// TwinCAT 3 PLC project ButtonControlledGarageDoor
// ProgramVersion: 3.1.4024.0
// libraries:
//   Tc2_Standard, * (Beckhoff Automation GmbH)
//   Tc2_System, * (Beckhoff Automation GmbH)
//   Tc3_Module, * (Beckhoff Automation GmbH)
//   VisuDialogs, * (System)
// project tree:
//   / GlobalTextList.TcGTLO, PlcTask.TcTTO, Visualization Manager.TcVMO (not stored)
//   POUs/ FB_DoorController.TcPOU, FB_BlinkingLight.TcPOU, MAIN.TcPOU
//   VISUs/ Visualization.TcVIS
// real-time tasks:
//   TASK PlcTask: cycle T#10ms, priority 20, ADS port 350

CONFIGURATION ButtonControlledGarageDoor
    RESOURCE PLC ON TwinCAT3
        TASK PlcTask(INTERVAL := T#10ms, PRIORITY := 20);
        PROGRAM MAIN WITH PlcTask : MAIN;
    END_RESOURCE
END_CONFIGURATION

// ---- POUs/MAIN.TcPOU
PROGRAM MAIN
VAR
	fbGarage1 : FB_DoorController;
	bActuation1 : BOOL;
	bOpenButton1 : BOOL;
	bCloseButton1 : BOOL;
	bDriveOverload1 : BOOL; 
	dwLightDelay1 : DWORD := 1000;
	dwBlinkingTimeOn1 : DWORD := 500;
	dwBlinkingTimeOff1 : DWORD := 250;
	bDoorLight1 : BOOL;
	bOpeningLight1 : BOOL;
	bClosingLight1 : BOOL;
	bNoError1 : BOOL;
	sErrorMessage1 : STRING;
	
	fbGarage2 : FB_DoorController;
	bActuation2 : BOOL;
	bOpenButton2 : BOOL;
	bCloseButton2 : BOOL;
	bDriveOverload2 : BOOL; 
	dwLightDelay2 : DWORD := 1000;
	dwBlinkingTimeOn2 : DWORD := 500;
	dwBlinkingTimeOff2 : DWORD := 250;
	bDoorLight2 : BOOL;
	bOpeningLight2 : BOOL;
	bClosingLight2 : BOOL;
	bNoError2 : BOOL;
	sErrorMessage2 : STRING;
END_VAR

fbGarage1(bActuation := bActuation1, 
		  bOpenButton := bOpenButton1, 
		  bCloseButton := bCloseButton1, 
		  bDriveOverload := bDriveOverload1,
		  dwLightDelay := dwLightDelay1,
		  dwBlinkingTimeOn := dwBlinkingTimeOn1,
		  dwBlinkingTimeOff := dwBlinkingTimeOff1,
		  bDoorLight => bDoorLight1, 
		  bOpeningLight => bOpeningLight1, 
		  bClosingLight => bClosingLight1,
		  bNoError => bNoError1,
		  sErrorMessage => sErrorMessage1); 
		  
fbGarage2(bActuation := bActuation2, 
		  bOpenButton := bOpenButton2, 
		  bCloseButton := bCloseButton2, 
		  bDriveOverload := bDriveOverload2,
		  dwLightDelay := dwLightDelay2,
		  dwBlinkingTimeOn := dwBlinkingTimeOn2,
		  dwBlinkingTimeOff := dwBlinkingTimeOff2,
		  bDoorLight => bDoorLight2, 
		  bOpeningLight => bOpeningLight2, 
		  bClosingLight => bClosingLight2,
		  bNoError => bNoError2,
		  sErrorMessage => sErrorMessage2);

END_PROGRAM

// ---- POUs/FB_DoorController.TcPOU
FUNCTION_BLOCK FB_DoorController
VAR_INPUT
	// Button that starts the door
	bActuation : BOOL;
	
	// Buttons that open / close the door respectively
	bOpenButton: BOOL;
	bCloseButton : BOOL;
	
	// Button that makes the door go into a drive overload
	bDriveOverload : BOOL;
	
	// How much time (in ms) should pass in order for the light to turn off when the door has opened / closed 
	dwLightDelay : DWORD;
	
	// On/off times (in miliseconds) for when the garage door light is blinking in state of error
	dwBlinkingTimeOn : DWORD;
	dwBlinkingTimeOff : DWORD;
END_VAR
VAR_OUTPUT
	// Outputs sent to actuators stating that the door is moving up / down
	bDoorUp : BOOL;
	bDoorDown : BOOL;
	
	// Indicates whether the door light should be on or off
	bDoorLight : BOOL;
	
	// Lights that turn on if the door is opened / closed
	bOpeningLight : BOOL;
	bClosingLight : BOOL;
	
	// Variable that'll tell me if I'm in an error state or not
	bNoError : BOOL := TRUE;
	// Displaying a message according to the error we are encountering
	sErrorMessage : STRING;
END_VAR
VAR
	// Variables stating whether the door is opened or closed
	bDoorOpen : BOOL;
	bDoorClosed : BOOL := TRUE;	// Assumption that in the beginning the door is closed
	
	// TRUE when the process was paused during opening / closing
	bPauseWhenOpening : BOOL;
	bPauseWhenClosing : BOOL;

	(* Timer needed for turning the door light off after a certain period of time passes 
	after the door has been opened / closed *)
	fbLightTimer : TON;
	
	// Trigger functions to deal with bouncing
	fbActuation : R_TRIG;
	fbOpenButton : R_TRIG;
	fbCloseButton : R_TRIG;
	fbDriveOverloadButton : R_TRIG;
	
	(* Instance of the BlinkingLight FB needed for the blinking of the actuation button 
	when it goes to an error state *)
	fbBlinkingLight : FB_BlinkingLight;
	
	// Variable needed for initializing the CASE structure states
	nCurrentState : DINT;
	
	// Variables stating which errors we are encountering
	bDriveError : BOOL;
	bOpenError : BOOL; 
	bCloseError : BOOL;
	
	(* Temporary variable that helps me overcome a problem I'm facing due to
	   bOpenButton and bCloseButton being tappers *)
	bPom : BOOL;
	
	// Variables needed only for the visualisation
	Rect1 : BOOL;
	Rect2 : BOOL;

END_VAR

(* This FB is intended to manage the operation of a garage door. It processes inputs
   from various buttons (bActuation, bOpenButton, bCloseButton) and it handles drive
   overloads (bDriveOverload). The block controls the movement of the door (bDoorUp,
   bDoorDown), the activation of lights (bDoorLight, bOpeningLight, bClosingLight),
   and transitions between different states (idle, opening, closing, error). The FB
   also manages the timing for the door's lights, espeially when they need to blink
   in case of errors. Additionally, it tracks whether the door is fully opened or
   fully closed, handles pauses during opening or closing, and displays error messages
   when needed. *)

// Rising edge logic in order to stop bouncing (the signal persisting longer than intended)
fbActuation(CLK := bActuation);
bActuation := fbActuation.Q;
fbOpenButton(CLK := bOpenButton);
bOpenButton := fbOpenButton.Q;
fbCloseButton(CLK := bCloseButton);
bCloseButton := fbCloseButton.Q;
fbDriveOverloadButton(CLK := bDriveOverload);
bDriveOverload := fbDriveOverloadButton.Q;

CASE nCurrentState OF
	
	0:	// Idle
	(* The door is at rest. If the actuation button is pressed, the door either opens 
	   (if closed) or closes (if open). It also checks for a drive overload to 
	   transition into an error state. *)
	
	// If the overload sensor is activated, go to the error state
	IF bDriveOverload THEN
		nCurrentState := 999;
	END_IF
	
	// Reseting
	fbLightTimer.IN := FALSE;
	bDoorLight := FALSE;
	bOpeningLight := FALSE;
	bClosingLight := FALSE;
	
	// If the actuation button is pressed and the door is closed -> open it
	IF bActuation AND (bDoorClosed OR bPauseWhenClosing) THEN
		nCurrentState := 100;
	// If the actuation button is pressed and the door is opened -> close it
	ELSIF bActuation AND (bDoorOpen OR bPauseWhenOpening) THEN
		nCurrentState := 200;
	END_IF
	
	100:	// Opening
	(* The door is moving upwards. It activates the appropriate light and monitors for
	   errors like drive overload or the close button being pressed. If the door reaches 
	   the fully open position, it sets the bDoorOpen flag to TRUE, stops the opening 
	   process, and returns to the idle state. If an error occurs, it pauses the opening 
	   and transitions to the error state. *)
	
	(* If the overload sensor is activated or if the close button is pressed, go to the error state. 
	   bPauseWhenClosing is true because I want to continue with opening after I get out of the error state *)
	IF bDriveOverload OR bCloseButton THEN
		IF bDriveOverload THEN
			bdriveError := TRUE;	
		ELSIF bCloseButton THEN
			bCloseError := TRUE;
		END_IF
		
		bPauseWhenOpening := FALSE;
		bPauseWhenClosing := TRUE;
		nCurrentState := 999;
	END_IF
	
	// RESET EVERYTHING THAT'S GOTTA DO WITH CLOSING HERE
	bDoorDown := FALSE;
	bDoorClosed := FALSE;
	
	// State that the door should go up and turn the light on
	bDoorUp := TRUE;
	bDoorLight := TRUE;
	bOpeningLight := TRUE;
	
	// Code needed only for the visualisation
	Rect1 := TRUE;
	
	// Logic for opening
	IF bOpenButton OR bPom THEN	
		bPom := TRUE;
		bDoorOpen := TRUE;
		bPauseWhenClosing := FALSE;
		bOpeningLight := FALSE;
		
		Rect2 := TRUE;	// Needed only for the visualization
		
		fbLightTimer.IN := TRUE;
		IF fbLightTimer.Q THEN
			bPom := FALSE;
			bDoorLight := FALSE;
			nCurrentState := 0;
		END_IF		
	END_IF
	
	// The opening is paused -> go to idle state
	IF bActuation THEN
		bPauseWhenOpening := TRUE;
		bPauseWhenClosing := FALSE;
		bOpeningLight := FALSE;
	END_IF
	
	IF bPauseWhenOpening THEN
		fbLightTimer.IN := TRUE;
			IF fbLightTimer.Q THEN
				bDoorLight := FALSE;
				nCurrentState := 0;
			END_IF
	END_IF
	
	200:	// Closing
	(* The door is moving downwards. It manages the closing light and checks for errors
	   such as the open button being pressed or a drive overload. If the door reaches the 
	   fully closed position, it sets the bDoorClosed flag to TRUE, stops the closing 
	   process, and returns to the idle state. Similar to the opening state, any error 
	   pauses the closing process and transitions to the error state. *)
	
	(* If the overload sensor is activated or if the open button is pressed, go to the error state. 
	   bPauseWhenOpening is true because I want to continue with closing after I get out of the error state *)
	IF bDriveOverload OR bOpenButton THEN
		IF bDriveOverload THEN
			bdriveError := TRUE;	
		ELSIF bOpenButton THEN
			bOpenError := TRUE;
		END_IF
		
		bPauseWhenOpening := TRUE;
		bPauseWhenClosing := FALSE;
		nCurrentState := 999;
	END_IF
	
	// RESET EVERYTHING THAT'S GOTTA DO WITH OPENING HERE
	bDoorUp := FALSE;
	bDoorOpen := FALSE;
	
	// State that the door should go down and turn the light on
	bDoorDown := TRUE;
	bDoorLight := TRUE;
	bClosingLight := TRUE;
	
	// Code needed only for the visualisation
	Rect2 := FALSE;
	
	// Logic for closing
	IF bCloseButton OR bPom THEN
		bPom := TRUE;
		bDoorClosed := TRUE;
		bPauseWhenOpening := FALSE;
		bClosingLight := FALSE;
		
		Rect1 := FALSE;	// Needed only for the visualization
		
		fbLightTimer.IN := TRUE;
		IF fbLightTimer.Q THEN
			bPom := FALSE;
			bDoorLight := FALSE;
			nCurrentState := 0;
		END_IF
	END_IF
	
	// The closing is paused -> go to idle state
	IF bActuation THEN
		bPauseWhenClosing := TRUE;
		bPauseWhenOpening := FALSE;
		bClosingLight := FALSE;
	END_IF
	
	IF bPauseWhenClosing THEN
		fbLightTimer.IN := TRUE;
			IF fbLightTimer.Q THEN
				bDoorLight := FALSE;
				nCurrentState := 0;
			END_IF
	END_IF
	
	999:	// Error
	(* The system has detected an error, such as a drive overload or conflicting 
	   open/close commands. The door movement stops, and the light blinks to indicate 
	   the error. The state persists until the actuation button is pressed again, 
	   resetting the system and returning to idle. Error messages are displayed based 
	   on the specific error encountered. *)
	
	bNoError := FALSE;
	
	IF bActuation THEN
		bNoError := TRUE;
		nCurrentState := 0;
	END_IF
	
	fbBlinkingLight(dwTimeOn :=  dwBlinkingTimeOn, dwTimeOff := dwBlinkingTimeOff, bLight => bDoorLight);
	
	// WRITE LOGIC TO STOP THE WHOLE PROCESS HERE (RESET EVERYTHING)
	bDoorUp := FALSE;
	bDoorDown := FALSE;
	
	// Write error messages for the appropriate errors
	IF bDriveError THEN
		bDriveError := FALSE;
		sErrorMessage := 'Error ID XXXX: Drive overload!';
	END_IF
	
	IF bOpenError THEN
		bOpenError := FALSE;
		sErrorMessage := 'Error ID XXXX: Trying to open the door while it is in a process of closing!';
	END_IF
	
	IF bCloseError THEN
		bCloseError := FALSE;
		sErrorMessage := 'Error ID XXXX: Trying to close the door while it is in a process of opening!';
	END_IF
	
END_CASE

fbLightTimer(PT := TO_TIME(dwLightDelay));

END_FUNCTION_BLOCK

// ---- POUs/FB_BlinkingLight.TcPOU
FUNCTION_BLOCK FB_BlinkingLight
VAR_INPUT
	dwTimeOn : DWORD;
	dwTimeOff : DWORD;
END_VAR
VAR_OUTPUT
	bLight : BOOL;	// Determines whether the light will be ON or OFF
END_VAR
VAR
	fbTimerOn : TON;
	fbTimerOff : TON;
	fbStartTrigger : R_TRIG;
	
	nCurrentPhase : INT := 10;	// 10 - ON, 20 - OFF
	
	bIsBlinking : bool;
END_VAR

CASE nCurrentPhase OF
    10:	// ON
        fbTimerOn(IN := TRUE, PT := DWORD_TO_TIME(dwTimeOn));
        IF fbTimerOn.Q THEN
            fbTimerOn(IN := FALSE); // Reset the on timer
            nCurrentPhase := 20;  // Move to the off phase
        END_IF
        bLight := TRUE;

    20:	// OFF
        fbTimerOff(IN := TRUE, PT := DWORD_TO_TIME(dwTimeOff));
        IF fbTimerOff.Q THEN
            fbTimerOff(IN := FALSE); // Reset the off timer
            nCurrentPhase := 10;  // Move to the On phase
        END_IF
        bLight := FALSE;
		
ELSE
	fbTimerOn(IN := FALSE);
    fbTimerOff(IN := FALSE);
    bLight := FALSE;
END_CASE

END_FUNCTION_BLOCK

// ---- GlobalTextList.TcGTLO
TEXTLIST GlobalTextList
  364 = '%d : %s'
  611 = '%s'
  888 = 'Actuation'
  773 = 'Change blinking off time'
  642 = 'Change blinking on time'
  147 = 'Change light delay time'
  954 = 'Close'
  193 = 'Drive overload'
  949 = 'Garage 1'
  16 = 'Garage 2'
  657 = 'Open'
END_TEXTLIST

// ---- VISUs/Visualization.TcVIS
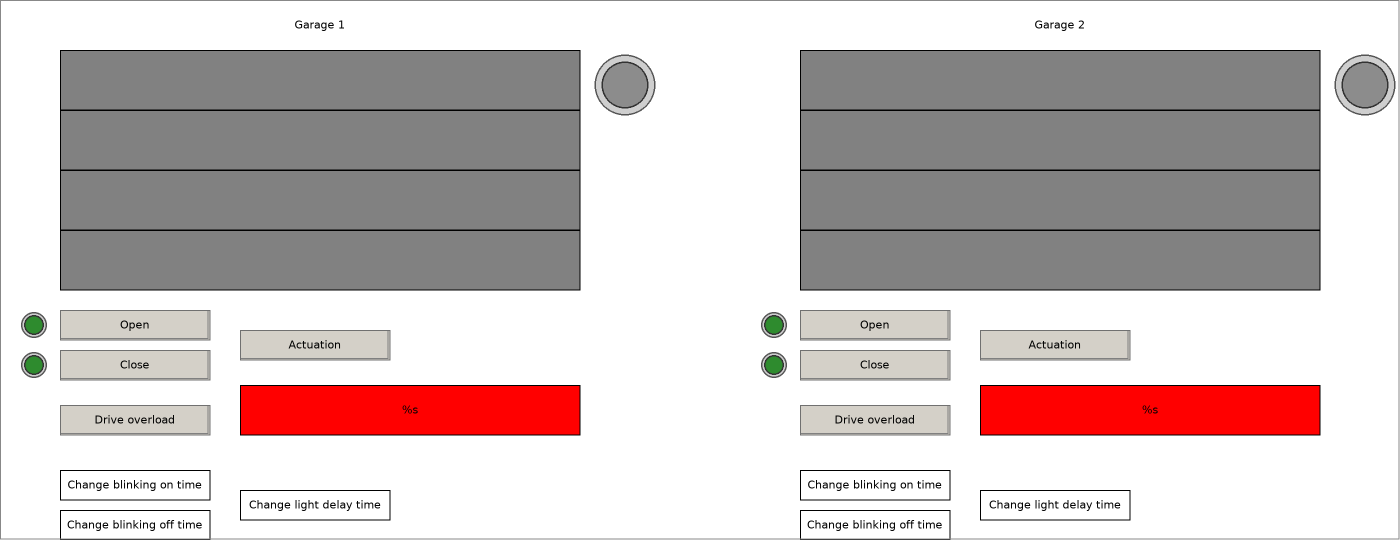
VISUALIZATION Visualization  // 1400x540
    Rectangle (60,50 520x240)
    Rectangle (60,50 520x60), invisible if: MAIN.fbGarage1.Rect2
    Button (240,330 150x30), "Actuation"
        tap MAIN.bActuation1
    Button (60,310 150x30), "Open"
        tap MAIN.bOpenButton1
    Button (60,350 150x30), "Close"
        tap MAIN.bCloseButton1
    Lamp1 (590,50 70x70), variable: MAIN.bDoorLight1, style: Lamp-Lamp1-Gray
    Lamp1 (19,310 30x30), variable: MAIN.bOpeningLight1, style: Lamp-Lamp1-Green
    Lamp1 (19,350 30x30), variable: MAIN.bClosingLight1, style: Lamp-Lamp1-Green
    Rectangle (60,110 520x60), invisible if: MAIN.fbGarage1.Rect2
    Rectangle (60,170 520x60), invisible if: MAIN.fbGarage1.Rect1
    Rectangle (60,230 520x60), invisible if: MAIN.fbGarage1.Rect1
    Button (60,405 150x30), "Drive overload"
        tap MAIN.bDriveOverload1
    Rectangle (800,50 520x240)
    Rectangle (800,50 520x60), invisible if: MAIN.fbGarage2.Rect2
    Button (980,330 150x30), "Actuation"
        tap MAIN.bActuation2
    Button (800,310 150x30), "Open"
        tap MAIN.bOpenButton2
    Button (800,350 150x30), "Close"
        tap MAIN.bCloseButton2
    Lamp1 (1330,50 70x70), variable: MAIN.bDoorLight2, style: Lamp-Lamp1-Gray
    Lamp1 (759,310 30x30), variable: MAIN.bOpeningLight2, style: Lamp-Lamp1-Green
    Lamp1 (759,350 30x30), variable: MAIN.bClosingLight2, style: Lamp-Lamp1-Green
    Rectangle (800,110 520x60), invisible if: MAIN.fbGarage2.Rect2
    Rectangle (800,170 520x60), invisible if: MAIN.fbGarage2.Rect1
    Rectangle (800,230 520x60), invisible if: MAIN.fbGarage2.Rect1
    Button (800,405 150x30), "Drive overload"
        tap MAIN.bDriveOverload2
    Label (245,10 150x30), "Garage 1"
    Label (985,10 150x30), "Garage 2"
    Rectangle (240,385 340x50), "%s", text variable: MAIN.sErrorMessage1, invisible if: MAIN.bNoError1
    Rectangle (980,385 340x50), "%s", text variable: MAIN.sErrorMessage2, invisible if: MAIN.bNoError2
    Rectangle (240,490 150x30), "Change light delay time"
        OnMouseClick: write MAIN.dwLightDelay1 via Default
    Rectangle (60,470 150x30), "Change blinking on time"
        OnMouseClick: write MAIN.dwBlinkingTimeOn1 via Default
    Rectangle (60,510 150x30), "Change blinking off time"
        OnMouseClick: write MAIN.dwBlinkingTimeOff1 via Default
    Rectangle (800,470 150x30), "Change blinking on time"
        OnMouseClick: write MAIN.dwBlinkingTimeOn2 via Default
    Rectangle (800,510 150x30), "Change blinking off time"
        OnMouseClick: write MAIN.dwBlinkingTimeOff2 via Default
    Rectangle (980,490 150x30), "Change light delay time"
        OnMouseClick: write MAIN.dwLightDelay2 via Default
END_VISUALIZATION
